// TwinCAT 3 PLC project plc
// ProgramVersion: 3.1.4023.0
// libraries:
//   Tc2_Standard, * (Beckhoff Automation GmbH)
//   Tc2_System, * (Beckhoff Automation GmbH)
//   Tc2_Utilities, * (Beckhoff Automation GmbH)
//   Tc3_Module, * (Beckhoff Automation GmbH)
// project tree:
//   DUTs/ E_EventType.TcDUT, ST_Events.TcDUT (not stored)
//   / PlcTask.TcTTO (not stored)
//   POUs/ F_UpdateTimestamp.TcPOU (not stored), MAIN.TcPOU

// ---- DUTs/E_EventType.TcDUT
{attribute 'qualified_only'}
{attribute 'strict'}
TYPE E_EventType :
(
	Undefined := 0,
	Message := 1,
	Alarm := 2
);
END_TYPE

// ---- POUs/MAIN.TcPOU
PROGRAM MAIN
VAR
	stEventsMain : ST_Events;
	xFlag :   BOOL := FALSE;
END_VAR

IF NOT xFlag THEN
		F_UpdateTimestamp (stEventsMain);
		xFlag := TRUE;
END_IF

END_PROGRAM
